// TIA Portal V18 export
TYPE "UDT_AHUsStsDelay"
// stored: IsFailsafeCompliant false
   STRUCT
      cCnt : Array[1..3] of Byte;
      cCheckingUpTime : Array[1..3] of Byte;
      cPreheatingTime : Array[1..3] of Byte;
      cStartingTime : Array[1..3] of Byte;
      cStoppingTime : Array[1..3] of Byte;
      cWorkOnFullRecycleTime : Array[1..3] of Byte;
   END_STRUCT;
   // cCheckingUpTime[1..2] := 10;
   // cPreheatingTime[1..2] := 20;
   // cStartingTime[1..2] := 10;
   // cStoppingTime[1..2] := 10;
END_TYPE
